TYPE ST_router_service :
STRUCT
END_STRUCT
END_TYPE

(* stored: Version 1.1.0.1, ProductVersion 3.1.4026.18
   DUT ST_router_service: Id {f22d3810-884a-43ed-bb36-cd91de7b7731} *)
